// TIA Portal V18 export
DATA_BLOCK "WN_2AxisMain"   // DB34
VERSION : 0.1
// stored: AutoNumber true, DBAccessibleFromOPCUA true, InstanceOfName ER_WORD, InstanceOfType FB
"ER_WORD"
   // VAR_INPUT
   //    ignoreNewEr : Bool;
   //    ak : Bool;
   //    x0 : Bool;
   //    x1 : Bool;
   //    x2 : Bool;
   //    x3 : Bool;
   //    x4 : Bool;
   //    x5 : Bool;
   //    x6 : Bool;
   //    x7 : Bool;
   //    x8 : Bool;
   //    x9 : Bool;
   //    x10 : Bool;
   //    x11 : Bool;
   //    x12 : Bool;
   //    x13 : Bool;
   //    x14 : Bool;
   //    x15 : Bool;
   //    selfreset0 : Bool;
   //    selfreset1 : Bool;
   //    selfreset2 : Bool;
   //    selfreset3 : Bool;
   //    selfreset4 : Bool;
   //    selfreset5 : Bool;
   //    selfreset6 : Bool;
   //    selfreset7 : Bool;
   //    selfreset8 : Bool;
   //    selfreset9 : Bool;
   //    selfreset10 : Bool;
   //    selfreset11 : Bool;
   //    selfreset12 : Bool;
   //    selfreset13 : Bool;
   //    selfreset14 : Bool;
   //    selfreset15 : Bool;
   // END_VAR
   // VAR_OUTPUT
   //    _w : Word;
   //    er : Bool;
   //    count : Int;
   //    "a_er[0]" : Bool;
   //    "a_er[1]" : Bool;
   //    "a_er[2]" : Bool;
   //    "a_er[3]" : Bool;
   //    "a_er[4]" : Bool;
   //    "a_er[5]" : Bool;
   //    "a_er[6]" : Bool;
   //    "a_er[7]" : Bool;
   //    "a_er[8]" : Bool;
   //    "a_er[9]" : Bool;
   //    "a_er[10]" : Bool;
   //    "a_er[11]" : Bool;
   //    "a_er[12]" : Bool;
   //    "a_er[13]" : Bool;
   //    "a_er[14]" : Bool;
   //    "a_er[15]" : Bool;
   // END_VAR
   // VAR
   //    a_er : Array[0..15] of Bool;
   //    a_x : Array[0..15] of Bool;
   //    a_is_self_reset : Array[0..15] of Bool;
   // END_VAR
BEGIN
END_DATA_BLOCK
